// TIA Portal V17 export
// export: Created 2025-03-13T10:30:04.4591601Z, ExportSetting WithDefaults, DisplayName Totally Integrated Automation Portal, DisplayVersion V17 Update 8, DisplayName TIA Portal Openness, DisplayVersion V17 Update 8, DisplayName TIA Portal Version Control Interface, DisplayVersion V17, DisplayName SINAMICS Startdrive Advanced, DisplayVersion V17 SP2, DisplayName SINAMICS Startdrive G110M, G120, G120C, G120D, G120P, G115D, DisplayVersion V17 SP2, DisplayName SINAMICS Startdrive G130, G150, S120, S150, SINAMICS MV, S210, DisplayVersion V17 SP2, DisplayName STEP 7 Professional, DisplayVersion V17 Update 8, DisplayName SINUMERIK ONE STEP 7 Toolbox, DisplayVersion V17 Update 12, DisplayName SINUMERIK 840D sl STEP 7 Toolbox, DisplayVersion V17 Update 12, DisplayName STEP 7 Safety, DisplayVersion V17 Update 6, DisplayName WinCC Advanced, DisplayVersion V17 Update 8
FUNCTION "FC2120_MPP_ITC_IPC" : Void   // FC2120, LAD
{ S7_Optimized_Access := 'FALSE' }
AUTHOR : ETXETAR
VERSION : 1.0
// stored: AutoNumber false, IsIECCheckEnabled false, SetENOAutomatically false, UDAEnableTagReadback false
   VAR_TEMP
      O_BYTE_0 : Struct   // OPTIONS BYTE 0
         IPC : Bool;   // IPC OPTION
      END_STRUCT;
      TCU_INDEX_SEL : Int;
   END_VAR
   VAR CONSTANT
      FC_NUMBER : DInt := 2120;   // FC NUMBER
   END_VAR
   VAR_TEMP   // added for the SCL form of the ladder/FBD networks
      _w1 : Bool;
      _w2 : Bool;
   END_VAR
BEGIN

REGION Network 1: OPTIONS
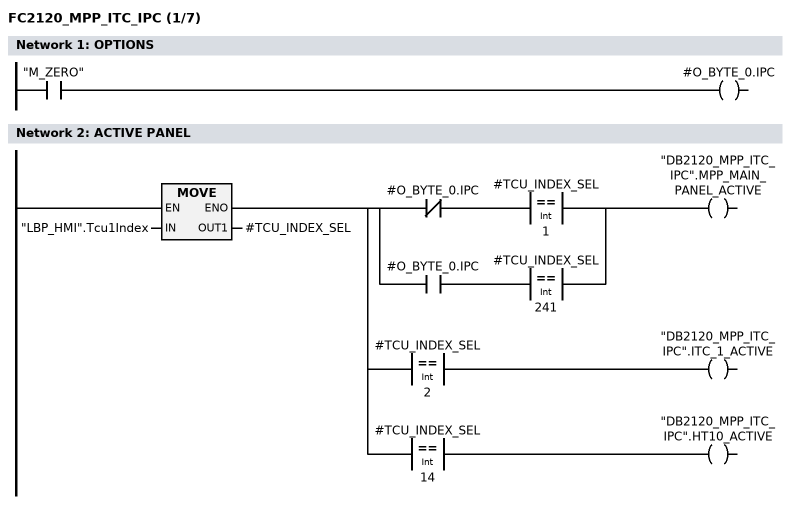
   RUNG wire#powerrail
      Contact( "M_ZERO" )
      Coil( #O_BYTE_0.IPC )
   END_RUNG
   // the same network as SCL:
   #O_BYTE_0.IPC := "M_ZERO";
END_REGION

REGION Network 2: ACTIVE PANEL
   RUNG wire#powerrail
      { S7_GenerateENO := "TRUE" } Move(in := "LBP_HMI".Tcu1Index, out1 => #TCU_INDEX_SEL)
      wire#w1
      I_Contact( #O_BYTE_0.IPC )
      { S7_Templates := "SrcType := Int" } EQ_Contact(in1 := #TCU_INDEX_SEL, in2 := 1)
      wire#w2
      Coil( "DB2120_MPP_ITC_IPC".MPP_MAIN_PANEL_ACTIVE )
   END_RUNG
   RUNG wire#w1
      Contact( #O_BYTE_0.IPC )
      { S7_Templates := "SrcType := Int" } EQ_Contact(in1 := #TCU_INDEX_SEL, in2 := 241)
   END_RUNG wire#w2
   RUNG wire#w1
      { S7_Templates := "SrcType := Int" } EQ_Contact(in1 := #TCU_INDEX_SEL, in2 := 2)
      Coil( "DB2120_MPP_ITC_IPC".ITC_1_ACTIVE )
   END_RUNG
   RUNG wire#w1
      { S7_Templates := "SrcType := Int" } EQ_Contact(in1 := #TCU_INDEX_SEL, in2 := 14)
      Coil( "DB2120_MPP_ITC_IPC".HT10_ACTIVE )
   END_RUNG
   // the same network as SCL:
   // ENO of a box is taken as its EN; it also drops when the box reports an error
   #TCU_INDEX_SEL := "LBP_HMI".Tcu1Index;
   "DB2120_MPP_ITC_IPC".MPP_MAIN_PANEL_ACTIVE := (NOT #O_BYTE_0.IPC AND (#TCU_INDEX_SEL = 1)) OR (#O_BYTE_0.IPC AND (#TCU_INDEX_SEL = 241));
   "DB2120_MPP_ITC_IPC".ITC_1_ACTIVE := #TCU_INDEX_SEL = 2;
   "DB2120_MPP_ITC_IPC".HT10_ACTIVE := #TCU_INDEX_SEL = 14;
END_REGION

REGION Network 3: OVERRIDE
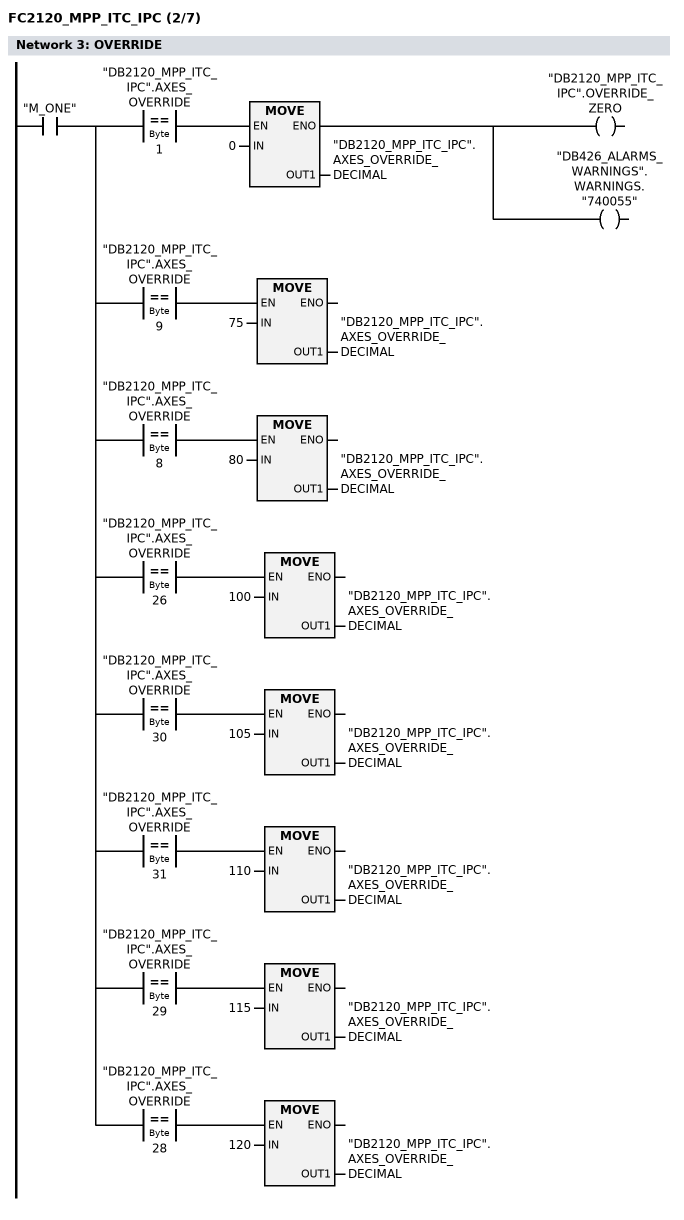
   RUNG wire#powerrail
      Contact( "M_ONE" )
      wire#w1
      { S7_Templates := "SrcType := Byte" } EQ_Contact(in1 := "DB2120_MPP_ITC_IPC".AXES_OVERRIDE, in2 := 1)
      { S7_GenerateENO := "TRUE" } Move(in := 0, out1 => "DB2120_MPP_ITC_IPC".AXES_OVERRIDE_DECIMAL)
      wire#w2
      Coil( "DB2120_MPP_ITC_IPC".OVERRIDE_ZERO )
   END_RUNG
   RUNG wire#w2
      Coil( "DB426_ALARMS_WARNINGS".WARNINGS."740055" )
   END_RUNG
   RUNG wire#w1
      { S7_Templates := "SrcType := Byte" } EQ_Contact(in1 := "DB2120_MPP_ITC_IPC".AXES_OVERRIDE, in2 := 9)
      { S7_GenerateENO := "TRUE" } Move(in := 75, out1 => "DB2120_MPP_ITC_IPC".AXES_OVERRIDE_DECIMAL)
   END_RUNG
   RUNG wire#w1
      { S7_Templates := "SrcType := Byte" } EQ_Contact(in1 := "DB2120_MPP_ITC_IPC".AXES_OVERRIDE, in2 := 8)
      { S7_GenerateENO := "TRUE" } Move(in := 80, out1 => "DB2120_MPP_ITC_IPC".AXES_OVERRIDE_DECIMAL)
   END_RUNG
   RUNG wire#w1
      { S7_Templates := "SrcType := Byte" } EQ_Contact(in1 := "DB2120_MPP_ITC_IPC".AXES_OVERRIDE, in2 := 26)
      { S7_GenerateENO := "TRUE" } Move(in := 100, out1 => "DB2120_MPP_ITC_IPC".AXES_OVERRIDE_DECIMAL)
   END_RUNG
   RUNG wire#w1
      { S7_Templates := "SrcType := Byte" } EQ_Contact(in1 := "DB2120_MPP_ITC_IPC".AXES_OVERRIDE, in2 := 30)
      { S7_GenerateENO := "TRUE" } Move(in := 105, out1 => "DB2120_MPP_ITC_IPC".AXES_OVERRIDE_DECIMAL)
   END_RUNG
   RUNG wire#w1
      { S7_Templates := "SrcType := Byte" } EQ_Contact(in1 := "DB2120_MPP_ITC_IPC".AXES_OVERRIDE, in2 := 31)
      { S7_GenerateENO := "TRUE" } Move(in := 110, out1 => "DB2120_MPP_ITC_IPC".AXES_OVERRIDE_DECIMAL)
   END_RUNG
   RUNG wire#w1
      { S7_Templates := "SrcType := Byte" } EQ_Contact(in1 := "DB2120_MPP_ITC_IPC".AXES_OVERRIDE, in2 := 29)
      { S7_GenerateENO := "TRUE" } Move(in := 115, out1 => "DB2120_MPP_ITC_IPC".AXES_OVERRIDE_DECIMAL)
   END_RUNG
   RUNG wire#w1
      { S7_Templates := "SrcType := Byte" } EQ_Contact(in1 := "DB2120_MPP_ITC_IPC".AXES_OVERRIDE, in2 := 28)
      { S7_GenerateENO := "TRUE" } Move(in := 120, out1 => "DB2120_MPP_ITC_IPC".AXES_OVERRIDE_DECIMAL)
   END_RUNG
   // the same network as SCL:
   // ENO of a box is taken as its EN; it also drops when the box reports an error
   #_w1 := "M_ONE" AND ("DB2120_MPP_ITC_IPC".AXES_OVERRIDE = 1);
   IF #_w1 THEN "DB2120_MPP_ITC_IPC".AXES_OVERRIDE_DECIMAL := 0; END_IF;
   "DB2120_MPP_ITC_IPC".OVERRIDE_ZERO := #_w1;
   "DB426_ALARMS_WARNINGS".WARNINGS."740055" := #_w1;
   IF "M_ONE" AND ("DB2120_MPP_ITC_IPC".AXES_OVERRIDE = 9) THEN
       "DB2120_MPP_ITC_IPC".AXES_OVERRIDE_DECIMAL := 75;
   END_IF;
   IF "M_ONE" AND ("DB2120_MPP_ITC_IPC".AXES_OVERRIDE = 8) THEN
       "DB2120_MPP_ITC_IPC".AXES_OVERRIDE_DECIMAL := 80;
   END_IF;
   IF "M_ONE" AND ("DB2120_MPP_ITC_IPC".AXES_OVERRIDE = 26) THEN
       "DB2120_MPP_ITC_IPC".AXES_OVERRIDE_DECIMAL := 100;
   END_IF;
   IF "M_ONE" AND ("DB2120_MPP_ITC_IPC".AXES_OVERRIDE = 30) THEN
       "DB2120_MPP_ITC_IPC".AXES_OVERRIDE_DECIMAL := 105;
   END_IF;
   IF "M_ONE" AND ("DB2120_MPP_ITC_IPC".AXES_OVERRIDE = 31) THEN
       "DB2120_MPP_ITC_IPC".AXES_OVERRIDE_DECIMAL := 110;
   END_IF;
   IF "M_ONE" AND ("DB2120_MPP_ITC_IPC".AXES_OVERRIDE = 29) THEN
       "DB2120_MPP_ITC_IPC".AXES_OVERRIDE_DECIMAL := 115;
   END_IF;
   IF "M_ONE" AND ("DB2120_MPP_ITC_IPC".AXES_OVERRIDE = 28) THEN
       "DB2120_MPP_ITC_IPC".AXES_OVERRIDE_DECIMAL := 120;
   END_IF;
END_REGION

REGION Network 4: OVERRIDE LOWER THAN 80
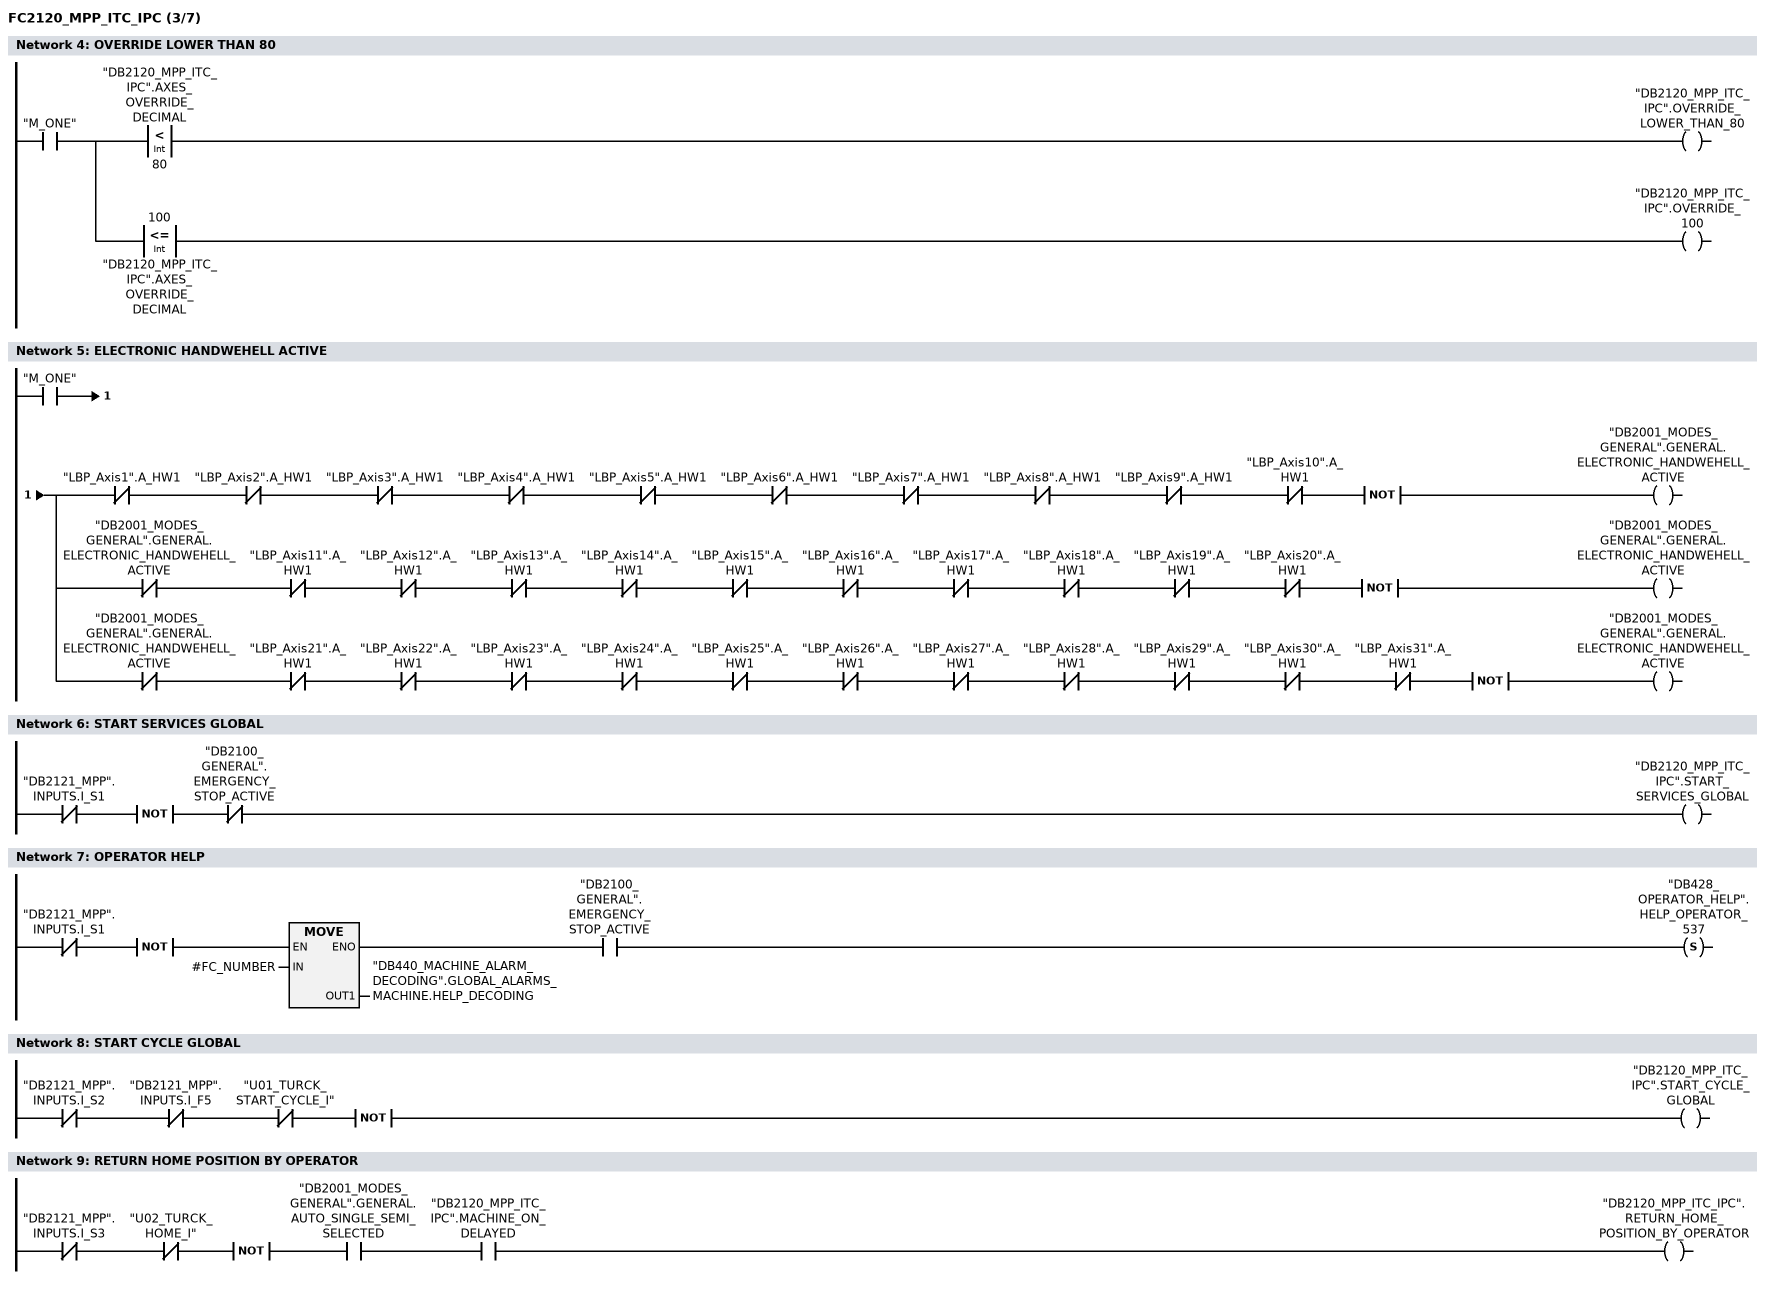
   RUNG wire#powerrail
      Contact( "M_ONE" )
      wire#w1
      { S7_Templates := "SrcType := Int" } LT_Contact(in1 := "DB2120_MPP_ITC_IPC".AXES_OVERRIDE_DECIMAL, in2 := 80)
      Coil( "DB2120_MPP_ITC_IPC".OVERRIDE_LOWER_THAN_80 )
   END_RUNG
   RUNG wire#w1
      { S7_Templates := "SrcType := Int" } LE_Contact(in1 := 100, in2 := "DB2120_MPP_ITC_IPC".AXES_OVERRIDE_DECIMAL)
      Coil( "DB2120_MPP_ITC_IPC".OVERRIDE_100 )
   END_RUNG
   // the same network as SCL:
   "DB2120_MPP_ITC_IPC".OVERRIDE_LOWER_THAN_80 := "M_ONE" AND ("DB2120_MPP_ITC_IPC".AXES_OVERRIDE_DECIMAL < 80);
   "DB2120_MPP_ITC_IPC".OVERRIDE_100 := "M_ONE" AND (100 <= "DB2120_MPP_ITC_IPC".AXES_OVERRIDE_DECIMAL);
END_REGION

REGION Network 5: ELECTRONIC HANDWEHELL ACTIVE
   RUNG wire#powerrail
      Contact( "M_ONE" )
      wire#w1
      I_Contact( "LBP_Axis1".A_HW1 )
      I_Contact( "LBP_Axis2".A_HW1 )
      I_Contact( "LBP_Axis3".A_HW1 )
      I_Contact( "LBP_Axis4".A_HW1 )
      I_Contact( "LBP_Axis5".A_HW1 )
      I_Contact( "LBP_Axis6".A_HW1 )
      I_Contact( "LBP_Axis7".A_HW1 )
      I_Contact( "LBP_Axis8".A_HW1 )
      I_Contact( "LBP_Axis9".A_HW1 )
      I_Contact( "LBP_Axis10".A_HW1 )
      Not()
      Coil( "DB2001_MODES_GENERAL".GENERAL.ELECTRONIC_HANDWEHELL_ACTIVE )
   END_RUNG
   RUNG wire#w1
      I_Contact( "DB2001_MODES_GENERAL".GENERAL.ELECTRONIC_HANDWEHELL_ACTIVE )
      I_Contact( "LBP_Axis11".A_HW1 )
      I_Contact( "LBP_Axis12".A_HW1 )
      I_Contact( "LBP_Axis13".A_HW1 )
      I_Contact( "LBP_Axis14".A_HW1 )
      I_Contact( "LBP_Axis15".A_HW1 )
      I_Contact( "LBP_Axis16".A_HW1 )
      I_Contact( "LBP_Axis17".A_HW1 )
      I_Contact( "LBP_Axis18".A_HW1 )
      I_Contact( "LBP_Axis19".A_HW1 )
      I_Contact( "LBP_Axis20".A_HW1 )
      Not()
      Coil( "DB2001_MODES_GENERAL".GENERAL.ELECTRONIC_HANDWEHELL_ACTIVE )
   END_RUNG
   RUNG wire#w1
      I_Contact( "DB2001_MODES_GENERAL".GENERAL.ELECTRONIC_HANDWEHELL_ACTIVE )
      I_Contact( "LBP_Axis21".A_HW1 )
      I_Contact( "LBP_Axis22".A_HW1 )
      I_Contact( "LBP_Axis23".A_HW1 )
      I_Contact( "LBP_Axis24".A_HW1 )
      I_Contact( "LBP_Axis25".A_HW1 )
      I_Contact( "LBP_Axis26".A_HW1 )
      I_Contact( "LBP_Axis27".A_HW1 )
      I_Contact( "LBP_Axis28".A_HW1 )
      I_Contact( "LBP_Axis29".A_HW1 )
      I_Contact( "LBP_Axis30".A_HW1 )
      I_Contact( "LBP_Axis31".A_HW1 )
      Not()
      Coil( "DB2001_MODES_GENERAL".GENERAL.ELECTRONIC_HANDWEHELL_ACTIVE )
   END_RUNG
   // the same network as SCL:
   "DB2001_MODES_GENERAL".GENERAL.ELECTRONIC_HANDWEHELL_ACTIVE := NOT ("M_ONE" AND NOT "LBP_Axis1".A_HW1 AND NOT "LBP_Axis2".A_HW1 AND NOT "LBP_Axis3".A_HW1 AND NOT "LBP_Axis4".A_HW1 AND NOT "LBP_Axis5".A_HW1 AND NOT "LBP_Axis6".A_HW1 AND NOT "LBP_Axis7".A_HW1 AND NOT "LBP_Axis8".A_HW1 AND NOT "LBP_Axis9".A_HW1 AND NOT "LBP_Axis10".A_HW1);
   "DB2001_MODES_GENERAL".GENERAL.ELECTRONIC_HANDWEHELL_ACTIVE := NOT ("M_ONE" AND NOT "DB2001_MODES_GENERAL".GENERAL.ELECTRONIC_HANDWEHELL_ACTIVE AND NOT "LBP_Axis11".A_HW1 AND NOT "LBP_Axis12".A_HW1 AND NOT "LBP_Axis13".A_HW1 AND NOT "LBP_Axis14".A_HW1 AND NOT "LBP_Axis15".A_HW1 AND NOT "LBP_Axis16".A_HW1 AND NOT "LBP_Axis17".A_HW1 AND NOT "LBP_Axis18".A_HW1 AND NOT "LBP_Axis19".A_HW1 AND NOT "LBP_Axis20".A_HW1);
   "DB2001_MODES_GENERAL".GENERAL.ELECTRONIC_HANDWEHELL_ACTIVE := NOT ("M_ONE" AND NOT "DB2001_MODES_GENERAL".GENERAL.ELECTRONIC_HANDWEHELL_ACTIVE AND NOT "LBP_Axis21".A_HW1 AND NOT "LBP_Axis22".A_HW1 AND NOT "LBP_Axis23".A_HW1 AND NOT "LBP_Axis24".A_HW1 AND NOT "LBP_Axis25".A_HW1 AND NOT "LBP_Axis26".A_HW1 AND NOT "LBP_Axis27".A_HW1 AND NOT "LBP_Axis28".A_HW1 AND NOT "LBP_Axis29".A_HW1 AND NOT "LBP_Axis30".A_HW1 AND NOT "LBP_Axis31".A_HW1);
END_REGION

REGION Network 6: START SERVICES GLOBAL
   RUNG wire#powerrail
      I_Contact( "DB2121_MPP".INPUTS.I_S1 )
      Not()
      I_Contact( "DB2100_GENERAL".EMERGENCY_STOP_ACTIVE )
      Coil( "DB2120_MPP_ITC_IPC".START_SERVICES_GLOBAL )
   END_RUNG
   // the same network as SCL:
   "DB2120_MPP_ITC_IPC".START_SERVICES_GLOBAL := NOT (NOT "DB2121_MPP".INPUTS.I_S1) AND NOT "DB2100_GENERAL".EMERGENCY_STOP_ACTIVE;
END_REGION

REGION Network 7: OPERATOR HELP
   RUNG wire#powerrail
      I_Contact( "DB2121_MPP".INPUTS.I_S1 )
      Not()
      { S7_GenerateENO := "TRUE" } Move(in := #FC_NUMBER, out1 => "DB440_MACHINE_ALARM_DECODING".GLOBAL_ALARMS_MACHINE.HELP_DECODING)
      Contact( "DB2100_GENERAL".EMERGENCY_STOP_ACTIVE )
      S_Coil( "DB428_OPERATOR_HELP".HELP_OPERATOR_537 )
   END_RUNG
   // the same network as SCL:
   // ENO of a box is taken as its EN; it also drops when the box reports an error
   #_w1 := NOT (NOT "DB2121_MPP".INPUTS.I_S1);
   IF #_w1 THEN "DB440_MACHINE_ALARM_DECODING".GLOBAL_ALARMS_MACHINE.HELP_DECODING := #FC_NUMBER; END_IF;
   IF #_w1 AND "DB2100_GENERAL".EMERGENCY_STOP_ACTIVE THEN
       "DB428_OPERATOR_HELP".HELP_OPERATOR_537 := TRUE;
   END_IF;
END_REGION

REGION Network 8: START CYCLE GLOBAL
   RUNG wire#powerrail
      I_Contact( "DB2121_MPP".INPUTS.I_S2 )
      I_Contact( "DB2121_MPP".INPUTS.I_F5 )
      I_Contact( "U01_TURCK_START_CYCLE_I" )
      Not()
      Coil( "DB2120_MPP_ITC_IPC".START_CYCLE_GLOBAL )
   END_RUNG
   // the same network as SCL:
   "DB2120_MPP_ITC_IPC".START_CYCLE_GLOBAL := NOT (NOT "DB2121_MPP".INPUTS.I_S2 AND NOT "DB2121_MPP".INPUTS.I_F5 AND NOT "U01_TURCK_START_CYCLE_I");
END_REGION

REGION Network 9: RETURN HOME POSITION BY OPERATOR
   RUNG wire#powerrail
      I_Contact( "DB2121_MPP".INPUTS.I_S3 )
      I_Contact( "U02_TURCK_HOME_I" )
      Not()
      Contact( "DB2001_MODES_GENERAL".GENERAL.AUTO_SINGLE_SEMI_SELECTED )
      Contact( "DB2120_MPP_ITC_IPC".MACHINE_ON_DELAYED )
      Coil( "DB2120_MPP_ITC_IPC".RETURN_HOME_POSITION_BY_OPERATOR )
   END_RUNG
   // the same network as SCL:
   "DB2120_MPP_ITC_IPC".RETURN_HOME_POSITION_BY_OPERATOR := NOT (NOT "DB2121_MPP".INPUTS.I_S3 AND NOT "U02_TURCK_HOME_I") AND "DB2001_MODES_GENERAL".GENERAL.AUTO_SINGLE_SEMI_SELECTED AND "DB2120_MPP_ITC_IPC".MACHINE_ON_DELAYED;
END_REGION

REGION Network 10: RETURN HOME POSITION FROM MPP-AUX PANEL
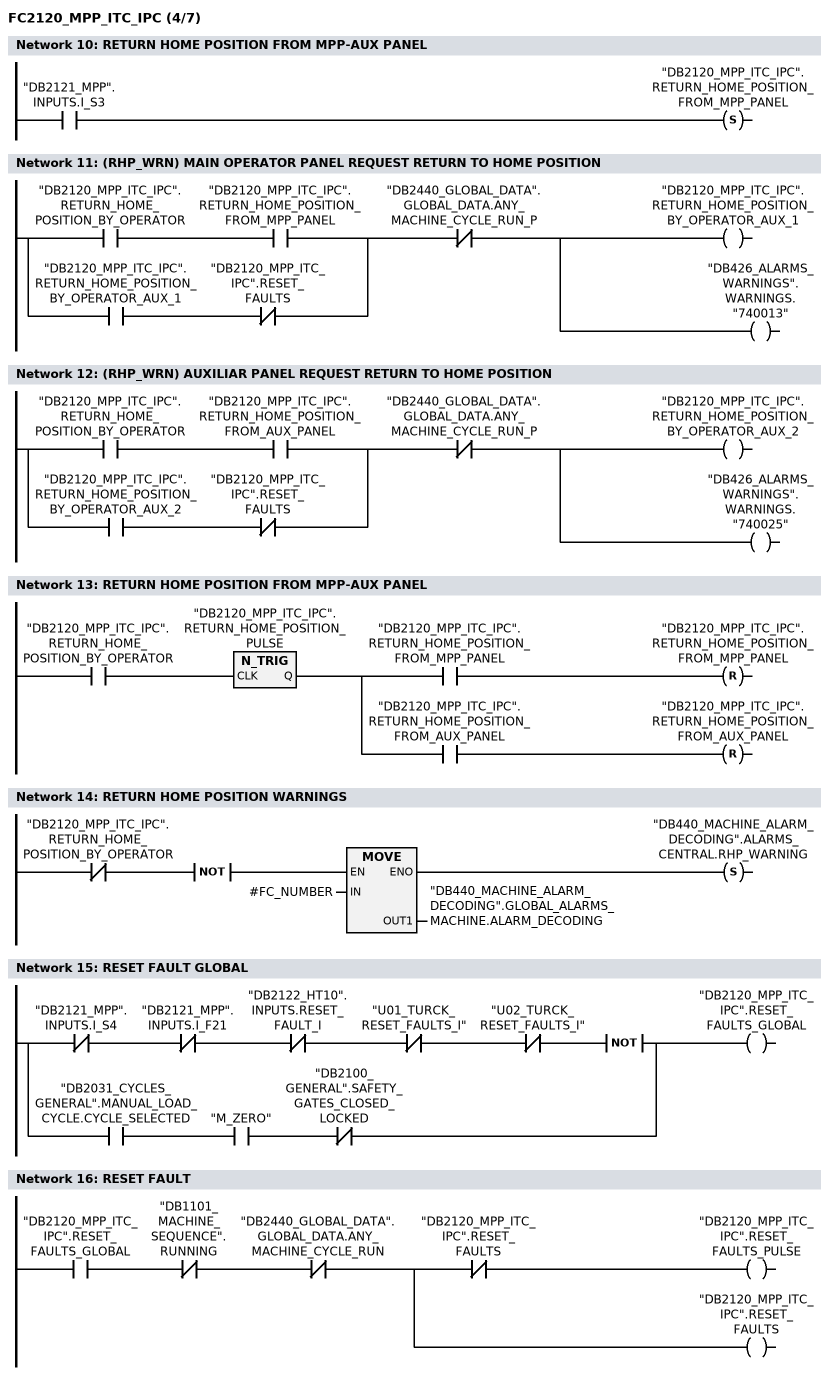
   RUNG wire#powerrail
      Contact( "DB2121_MPP".INPUTS.I_S3 )
      S_Coil( "DB2120_MPP_ITC_IPC".RETURN_HOME_POSITION_FROM_MPP_PANEL )
   END_RUNG
   // the same network as SCL:
   IF "DB2121_MPP".INPUTS.I_S3 THEN "DB2120_MPP_ITC_IPC".RETURN_HOME_POSITION_FROM_MPP_PANEL := TRUE; END_IF;
END_REGION

REGION Network 11: (RHP_WRN) MAIN OPERATOR PANEL REQUEST RETURN TO HOME POSITION
   RUNG wire#powerrail
      Contact( "DB2120_MPP_ITC_IPC".RETURN_HOME_POSITION_BY_OPERATOR )
      Contact( "DB2120_MPP_ITC_IPC".RETURN_HOME_POSITION_FROM_MPP_PANEL )
      wire#w1
      I_Contact( "DB2440_GLOBAL_DATA".GLOBAL_DATA.ANY_MACHINE_CYCLE_RUN_P )
      wire#w2
      Coil( "DB2120_MPP_ITC_IPC".RETURN_HOME_POSITION_BY_OPERATOR_AUX_1 )
   END_RUNG
   RUNG wire#powerrail
      Contact( "DB2120_MPP_ITC_IPC".RETURN_HOME_POSITION_BY_OPERATOR_AUX_1 )
      I_Contact( "DB2120_MPP_ITC_IPC".RESET_FAULTS )
   END_RUNG wire#w1
   RUNG wire#w2
      Coil( "DB426_ALARMS_WARNINGS".WARNINGS."740013" )
   END_RUNG
   // the same network as SCL:
   "DB2120_MPP_ITC_IPC".RETURN_HOME_POSITION_BY_OPERATOR_AUX_1 := (("DB2120_MPP_ITC_IPC".RETURN_HOME_POSITION_BY_OPERATOR AND "DB2120_MPP_ITC_IPC".RETURN_HOME_POSITION_FROM_MPP_PANEL) OR ("DB2120_MPP_ITC_IPC".RETURN_HOME_POSITION_BY_OPERATOR_AUX_1 AND NOT "DB2120_MPP_ITC_IPC".RESET_FAULTS)) AND NOT "DB2440_GLOBAL_DATA".GLOBAL_DATA.ANY_MACHINE_CYCLE_RUN_P;
   "DB426_ALARMS_WARNINGS".WARNINGS."740013" := "DB2120_MPP_ITC_IPC".RETURN_HOME_POSITION_BY_OPERATOR_AUX_1;
END_REGION

REGION Network 12: (RHP_WRN) AUXILIAR PANEL REQUEST RETURN TO HOME POSITION
   RUNG wire#powerrail
      Contact( "DB2120_MPP_ITC_IPC".RETURN_HOME_POSITION_BY_OPERATOR )
      Contact( "DB2120_MPP_ITC_IPC".RETURN_HOME_POSITION_FROM_AUX_PANEL )
      wire#w1
      I_Contact( "DB2440_GLOBAL_DATA".GLOBAL_DATA.ANY_MACHINE_CYCLE_RUN_P )
      wire#w2
      Coil( "DB2120_MPP_ITC_IPC".RETURN_HOME_POSITION_BY_OPERATOR_AUX_2 )
   END_RUNG
   RUNG wire#powerrail
      Contact( "DB2120_MPP_ITC_IPC".RETURN_HOME_POSITION_BY_OPERATOR_AUX_2 )
      I_Contact( "DB2120_MPP_ITC_IPC".RESET_FAULTS )
   END_RUNG wire#w1
   RUNG wire#w2
      Coil( "DB426_ALARMS_WARNINGS".WARNINGS."740025" )
   END_RUNG
   // the same network as SCL:
   "DB2120_MPP_ITC_IPC".RETURN_HOME_POSITION_BY_OPERATOR_AUX_2 := (("DB2120_MPP_ITC_IPC".RETURN_HOME_POSITION_BY_OPERATOR AND "DB2120_MPP_ITC_IPC".RETURN_HOME_POSITION_FROM_AUX_PANEL) OR ("DB2120_MPP_ITC_IPC".RETURN_HOME_POSITION_BY_OPERATOR_AUX_2 AND NOT "DB2120_MPP_ITC_IPC".RESET_FAULTS)) AND NOT "DB2440_GLOBAL_DATA".GLOBAL_DATA.ANY_MACHINE_CYCLE_RUN_P;
   "DB426_ALARMS_WARNINGS".WARNINGS."740025" := "DB2120_MPP_ITC_IPC".RETURN_HOME_POSITION_BY_OPERATOR_AUX_2;
END_REGION

REGION Network 13: RETURN HOME POSITION FROM MPP-AUX PANEL
   RUNG wire#powerrail
      Contact( "DB2120_MPP_ITC_IPC".RETURN_HOME_POSITION_BY_OPERATOR )
      N_Trig( "DB2120_MPP_ITC_IPC".RETURN_HOME_POSITION_PULSE )
      wire#w1
      Contact( "DB2120_MPP_ITC_IPC".RETURN_HOME_POSITION_FROM_MPP_PANEL )
      R_Coil( "DB2120_MPP_ITC_IPC".RETURN_HOME_POSITION_FROM_MPP_PANEL )
   END_RUNG
   RUNG wire#w1
      Contact( "DB2120_MPP_ITC_IPC".RETURN_HOME_POSITION_FROM_AUX_PANEL )
      R_Coil( "DB2120_MPP_ITC_IPC".RETURN_HOME_POSITION_FROM_AUX_PANEL )
   END_RUNG
   // the same network as SCL:
   #_w1 := NOT "DB2120_MPP_ITC_IPC".RETURN_HOME_POSITION_BY_OPERATOR AND "DB2120_MPP_ITC_IPC".RETURN_HOME_POSITION_PULSE;   // falling edge
   "DB2120_MPP_ITC_IPC".RETURN_HOME_POSITION_PULSE := "DB2120_MPP_ITC_IPC".RETURN_HOME_POSITION_BY_OPERATOR;
   IF #_w1 AND "DB2120_MPP_ITC_IPC".RETURN_HOME_POSITION_FROM_MPP_PANEL THEN
       "DB2120_MPP_ITC_IPC".RETURN_HOME_POSITION_FROM_MPP_PANEL := FALSE;
   END_IF;
   IF #_w1 AND "DB2120_MPP_ITC_IPC".RETURN_HOME_POSITION_FROM_AUX_PANEL THEN
       "DB2120_MPP_ITC_IPC".RETURN_HOME_POSITION_FROM_AUX_PANEL := FALSE;
   END_IF;
END_REGION

REGION Network 14: RETURN HOME POSITION WARNINGS
   RUNG wire#powerrail
      I_Contact( "DB2120_MPP_ITC_IPC".RETURN_HOME_POSITION_BY_OPERATOR )
      Not()
      { S7_GenerateENO := "TRUE" } Move(in := #FC_NUMBER, out1 => "DB440_MACHINE_ALARM_DECODING".GLOBAL_ALARMS_MACHINE.ALARM_DECODING)
      S_Coil( "DB440_MACHINE_ALARM_DECODING".ALARMS_CENTRAL.RHP_WARNING )
   END_RUNG
   // the same network as SCL:
   // ENO of a box is taken as its EN; it also drops when the box reports an error
   IF NOT (NOT "DB2120_MPP_ITC_IPC".RETURN_HOME_POSITION_BY_OPERATOR) THEN
       "DB440_MACHINE_ALARM_DECODING".GLOBAL_ALARMS_MACHINE.ALARM_DECODING := #FC_NUMBER;
       "DB440_MACHINE_ALARM_DECODING".ALARMS_CENTRAL.RHP_WARNING := TRUE;
   END_IF;
END_REGION

REGION Network 15: RESET FAULT GLOBAL
   RUNG wire#powerrail
      I_Contact( "DB2121_MPP".INPUTS.I_S4 )
      I_Contact( "DB2121_MPP".INPUTS.I_F21 )
      I_Contact( "DB2122_HT10".INPUTS.RESET_FAULT_I )
      I_Contact( "U01_TURCK_RESET_FAULTS_I" )
      I_Contact( "U02_TURCK_RESET_FAULTS_I" )
      Not()
      wire#w1
      Coil( "DB2120_MPP_ITC_IPC".RESET_FAULTS_GLOBAL )
   END_RUNG
   RUNG wire#powerrail
      Contact( "DB2031_CYCLES_GENERAL".MANUAL_LOAD_CYCLE.CYCLE_SELECTED )
      Contact( "M_ZERO" )
      I_Contact( "DB2100_GENERAL".SAFETY_GATES_CLOSED_LOCKED )
   END_RUNG wire#w1
   // the same network as SCL:
   "DB2120_MPP_ITC_IPC".RESET_FAULTS_GLOBAL := NOT (NOT "DB2121_MPP".INPUTS.I_S4 AND NOT "DB2121_MPP".INPUTS.I_F21 AND NOT "DB2122_HT10".INPUTS.RESET_FAULT_I AND NOT "U01_TURCK_RESET_FAULTS_I" AND NOT "U02_TURCK_RESET_FAULTS_I") OR ("DB2031_CYCLES_GENERAL".MANUAL_LOAD_CYCLE.CYCLE_SELECTED AND "M_ZERO" AND NOT "DB2100_GENERAL".SAFETY_GATES_CLOSED_LOCKED);
END_REGION

REGION Network 16: RESET FAULT
   RUNG wire#powerrail
      Contact( "DB2120_MPP_ITC_IPC".RESET_FAULTS_GLOBAL )
      I_Contact( "DB1101_MACHINE_SEQUENCE".RUNNING )
      I_Contact( "DB2440_GLOBAL_DATA".GLOBAL_DATA.ANY_MACHINE_CYCLE_RUN )
      wire#w1
      I_Contact( "DB2120_MPP_ITC_IPC".RESET_FAULTS )
      Coil( "DB2120_MPP_ITC_IPC".RESET_FAULTS_PULSE )
   END_RUNG
   RUNG wire#w1
      Coil( "DB2120_MPP_ITC_IPC".RESET_FAULTS )
   END_RUNG
   // the same network as SCL:
   #_w1 := "DB2120_MPP_ITC_IPC".RESET_FAULTS_GLOBAL AND NOT "DB1101_MACHINE_SEQUENCE".RUNNING AND NOT "DB2440_GLOBAL_DATA".GLOBAL_DATA.ANY_MACHINE_CYCLE_RUN;
   "DB2120_MPP_ITC_IPC".RESET_FAULTS_PULSE := #_w1 AND NOT "DB2120_MPP_ITC_IPC".RESET_FAULTS;
   "DB2120_MPP_ITC_IPC".RESET_FAULTS := #_w1;
END_REGION

REGION Network 17: STOP SERVICES GLOBAL
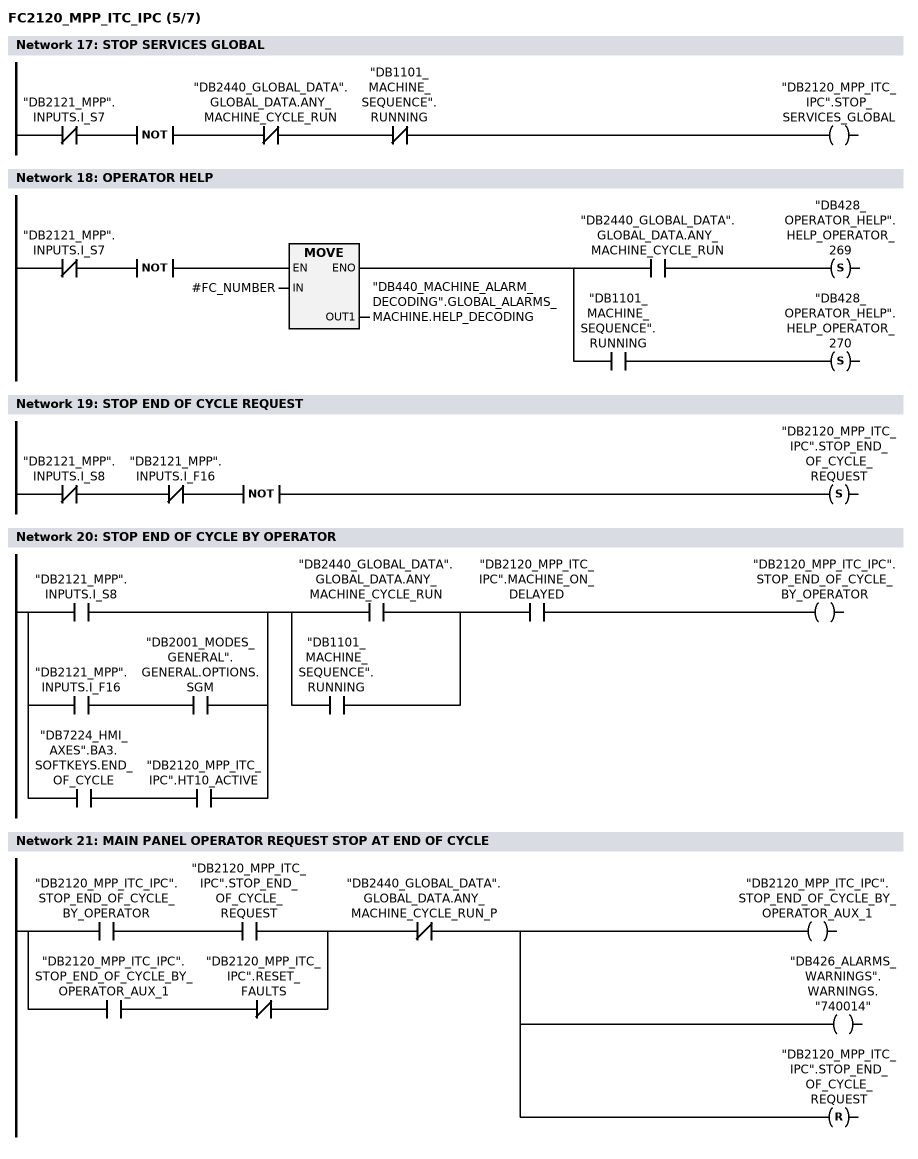
   RUNG wire#powerrail
      I_Contact( "DB2121_MPP".INPUTS.I_S7 )
      Not()
      I_Contact( "DB2440_GLOBAL_DATA".GLOBAL_DATA.ANY_MACHINE_CYCLE_RUN )
      I_Contact( "DB1101_MACHINE_SEQUENCE".RUNNING )
      Coil( "DB2120_MPP_ITC_IPC".STOP_SERVICES_GLOBAL )
   END_RUNG
   // the same network as SCL:
   "DB2120_MPP_ITC_IPC".STOP_SERVICES_GLOBAL := NOT (NOT "DB2121_MPP".INPUTS.I_S7) AND NOT "DB2440_GLOBAL_DATA".GLOBAL_DATA.ANY_MACHINE_CYCLE_RUN AND NOT "DB1101_MACHINE_SEQUENCE".RUNNING;
END_REGION

REGION Network 18: OPERATOR HELP
   RUNG wire#powerrail
      I_Contact( "DB2121_MPP".INPUTS.I_S7 )
      Not()
      { S7_GenerateENO := "TRUE" } Move(in := #FC_NUMBER, out1 => "DB440_MACHINE_ALARM_DECODING".GLOBAL_ALARMS_MACHINE.HELP_DECODING)
      wire#w1
      Contact( "DB2440_GLOBAL_DATA".GLOBAL_DATA.ANY_MACHINE_CYCLE_RUN )
      S_Coil( "DB428_OPERATOR_HELP".HELP_OPERATOR_269 )
   END_RUNG
   RUNG wire#w1
      Contact( "DB1101_MACHINE_SEQUENCE".RUNNING )
      S_Coil( "DB428_OPERATOR_HELP".HELP_OPERATOR_270 )
   END_RUNG
   // the same network as SCL:
   // ENO of a box is taken as its EN; it also drops when the box reports an error
   #_w1 := NOT (NOT "DB2121_MPP".INPUTS.I_S7);
   IF #_w1 THEN "DB440_MACHINE_ALARM_DECODING".GLOBAL_ALARMS_MACHINE.HELP_DECODING := #FC_NUMBER; END_IF;
   IF #_w1 AND "DB2440_GLOBAL_DATA".GLOBAL_DATA.ANY_MACHINE_CYCLE_RUN THEN
       "DB428_OPERATOR_HELP".HELP_OPERATOR_269 := TRUE;
   END_IF;
   IF #_w1 AND "DB1101_MACHINE_SEQUENCE".RUNNING THEN
       "DB428_OPERATOR_HELP".HELP_OPERATOR_270 := TRUE;
   END_IF;
END_REGION

REGION Network 19: STOP END OF CYCLE REQUEST
   RUNG wire#powerrail
      I_Contact( "DB2121_MPP".INPUTS.I_S8 )
      I_Contact( "DB2121_MPP".INPUTS.I_F16 )
      Not()
      S_Coil( "DB2120_MPP_ITC_IPC".STOP_END_OF_CYCLE_REQUEST )
   END_RUNG
   // the same network as SCL:
   IF NOT (NOT "DB2121_MPP".INPUTS.I_S8 AND NOT "DB2121_MPP".INPUTS.I_F16) THEN
       "DB2120_MPP_ITC_IPC".STOP_END_OF_CYCLE_REQUEST := TRUE;
   END_IF;
END_REGION

REGION Network 20: STOP END OF CYCLE BY OPERATOR
   RUNG wire#powerrail
      Contact( "DB2121_MPP".INPUTS.I_S8 )
      wire#w1
      Contact( "DB2440_GLOBAL_DATA".GLOBAL_DATA.ANY_MACHINE_CYCLE_RUN )
      wire#w2
      Contact( "DB2120_MPP_ITC_IPC".MACHINE_ON_DELAYED )
      Coil( "DB2120_MPP_ITC_IPC".STOP_END_OF_CYCLE_BY_OPERATOR )
   END_RUNG
   RUNG wire#powerrail
      Contact( "DB2121_MPP".INPUTS.I_F16 )
      Contact( "DB2001_MODES_GENERAL".GENERAL.OPTIONS.SGM )
   END_RUNG wire#w1
   RUNG wire#powerrail
      Contact( "DB7224_HMI_AXES".BA3.SOFTKEYS.END_OF_CYCLE )
      Contact( "DB2120_MPP_ITC_IPC".HT10_ACTIVE )
   END_RUNG wire#w1
   RUNG wire#w1
      Contact( "DB1101_MACHINE_SEQUENCE".RUNNING )
   END_RUNG wire#w2
   // the same network as SCL:
   "DB2120_MPP_ITC_IPC".STOP_END_OF_CYCLE_BY_OPERATOR := ("DB2121_MPP".INPUTS.I_S8 OR ("DB2121_MPP".INPUTS.I_F16 AND "DB2001_MODES_GENERAL".GENERAL.OPTIONS.SGM) OR ("DB7224_HMI_AXES".BA3.SOFTKEYS.END_OF_CYCLE AND "DB2120_MPP_ITC_IPC".HT10_ACTIVE)) AND ("DB2440_GLOBAL_DATA".GLOBAL_DATA.ANY_MACHINE_CYCLE_RUN OR "DB1101_MACHINE_SEQUENCE".RUNNING) AND "DB2120_MPP_ITC_IPC".MACHINE_ON_DELAYED;
END_REGION

REGION Network 21: MAIN PANEL OPERATOR REQUEST STOP AT END OF CYCLE
   RUNG wire#powerrail
      Contact( "DB2120_MPP_ITC_IPC".STOP_END_OF_CYCLE_BY_OPERATOR )
      Contact( "DB2120_MPP_ITC_IPC".STOP_END_OF_CYCLE_REQUEST )
      wire#w1
      I_Contact( "DB2440_GLOBAL_DATA".GLOBAL_DATA.ANY_MACHINE_CYCLE_RUN_P )
      wire#w2
      Coil( "DB2120_MPP_ITC_IPC".STOP_END_OF_CYCLE_BY_OPERATOR_AUX_1 )
   END_RUNG
   RUNG wire#powerrail
      Contact( "DB2120_MPP_ITC_IPC".STOP_END_OF_CYCLE_BY_OPERATOR_AUX_1 )
      I_Contact( "DB2120_MPP_ITC_IPC".RESET_FAULTS )
   END_RUNG wire#w1
   RUNG wire#w2
      Coil( "DB426_ALARMS_WARNINGS".WARNINGS."740014" )
   END_RUNG
   RUNG wire#w2
      R_Coil( "DB2120_MPP_ITC_IPC".STOP_END_OF_CYCLE_REQUEST )
   END_RUNG
   // the same network as SCL:
   "DB2120_MPP_ITC_IPC".STOP_END_OF_CYCLE_BY_OPERATOR_AUX_1 := (("DB2120_MPP_ITC_IPC".STOP_END_OF_CYCLE_BY_OPERATOR AND "DB2120_MPP_ITC_IPC".STOP_END_OF_CYCLE_REQUEST) OR ("DB2120_MPP_ITC_IPC".STOP_END_OF_CYCLE_BY_OPERATOR_AUX_1 AND NOT "DB2120_MPP_ITC_IPC".RESET_FAULTS)) AND NOT "DB2440_GLOBAL_DATA".GLOBAL_DATA.ANY_MACHINE_CYCLE_RUN_P;
   "DB426_ALARMS_WARNINGS".WARNINGS."740014" := "DB2120_MPP_ITC_IPC".STOP_END_OF_CYCLE_BY_OPERATOR_AUX_1;
   IF "DB2120_MPP_ITC_IPC".STOP_END_OF_CYCLE_BY_OPERATOR_AUX_1 THEN
       "DB2120_MPP_ITC_IPC".STOP_END_OF_CYCLE_REQUEST := FALSE;
   END_IF;
END_REGION

REGION Network 22: AUXILIARY PANEL OPERATOR REQUEST STOP AT END OF CYCLE
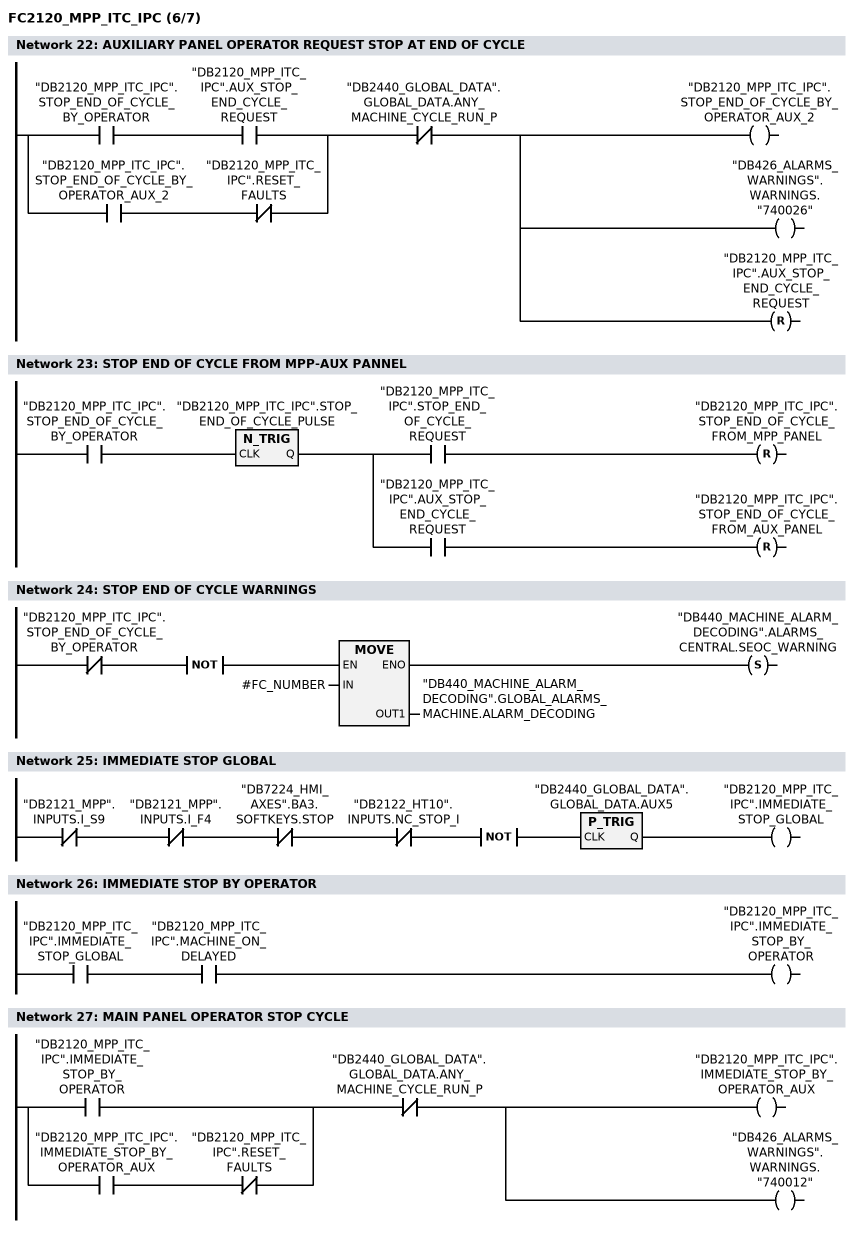
   RUNG wire#powerrail
      Contact( "DB2120_MPP_ITC_IPC".STOP_END_OF_CYCLE_BY_OPERATOR )
      Contact( "DB2120_MPP_ITC_IPC".AUX_STOP_END_CYCLE_REQUEST )
      wire#w1
      I_Contact( "DB2440_GLOBAL_DATA".GLOBAL_DATA.ANY_MACHINE_CYCLE_RUN_P )
      wire#w2
      Coil( "DB2120_MPP_ITC_IPC".STOP_END_OF_CYCLE_BY_OPERATOR_AUX_2 )
   END_RUNG
   RUNG wire#powerrail
      Contact( "DB2120_MPP_ITC_IPC".STOP_END_OF_CYCLE_BY_OPERATOR_AUX_2 )
      I_Contact( "DB2120_MPP_ITC_IPC".RESET_FAULTS )
   END_RUNG wire#w1
   RUNG wire#w2
      Coil( "DB426_ALARMS_WARNINGS".WARNINGS."740026" )
   END_RUNG
   RUNG wire#w2
      R_Coil( "DB2120_MPP_ITC_IPC".AUX_STOP_END_CYCLE_REQUEST )
   END_RUNG
   // the same network as SCL:
   "DB2120_MPP_ITC_IPC".STOP_END_OF_CYCLE_BY_OPERATOR_AUX_2 := (("DB2120_MPP_ITC_IPC".STOP_END_OF_CYCLE_BY_OPERATOR AND "DB2120_MPP_ITC_IPC".AUX_STOP_END_CYCLE_REQUEST) OR ("DB2120_MPP_ITC_IPC".STOP_END_OF_CYCLE_BY_OPERATOR_AUX_2 AND NOT "DB2120_MPP_ITC_IPC".RESET_FAULTS)) AND NOT "DB2440_GLOBAL_DATA".GLOBAL_DATA.ANY_MACHINE_CYCLE_RUN_P;
   "DB426_ALARMS_WARNINGS".WARNINGS."740026" := "DB2120_MPP_ITC_IPC".STOP_END_OF_CYCLE_BY_OPERATOR_AUX_2;
   IF "DB2120_MPP_ITC_IPC".STOP_END_OF_CYCLE_BY_OPERATOR_AUX_2 THEN
       "DB2120_MPP_ITC_IPC".AUX_STOP_END_CYCLE_REQUEST := FALSE;
   END_IF;
END_REGION

REGION Network 23: STOP END OF CYCLE FROM MPP-AUX PANNEL
   RUNG wire#powerrail
      Contact( "DB2120_MPP_ITC_IPC".STOP_END_OF_CYCLE_BY_OPERATOR )
      N_Trig( "DB2120_MPP_ITC_IPC".STOP_END_OF_CYCLE_PULSE )
      wire#w1
      Contact( "DB2120_MPP_ITC_IPC".STOP_END_OF_CYCLE_REQUEST )
      R_Coil( "DB2120_MPP_ITC_IPC".STOP_END_OF_CYCLE_FROM_MPP_PANEL )
   END_RUNG
   RUNG wire#w1
      Contact( "DB2120_MPP_ITC_IPC".AUX_STOP_END_CYCLE_REQUEST )
      R_Coil( "DB2120_MPP_ITC_IPC".STOP_END_OF_CYCLE_FROM_AUX_PANEL )
   END_RUNG
   // the same network as SCL:
   #_w1 := NOT "DB2120_MPP_ITC_IPC".STOP_END_OF_CYCLE_BY_OPERATOR AND "DB2120_MPP_ITC_IPC".STOP_END_OF_CYCLE_PULSE;   // falling edge
   "DB2120_MPP_ITC_IPC".STOP_END_OF_CYCLE_PULSE := "DB2120_MPP_ITC_IPC".STOP_END_OF_CYCLE_BY_OPERATOR;
   IF #_w1 AND "DB2120_MPP_ITC_IPC".STOP_END_OF_CYCLE_REQUEST THEN
       "DB2120_MPP_ITC_IPC".STOP_END_OF_CYCLE_FROM_MPP_PANEL := FALSE;
   END_IF;
   IF #_w1 AND "DB2120_MPP_ITC_IPC".AUX_STOP_END_CYCLE_REQUEST THEN
       "DB2120_MPP_ITC_IPC".STOP_END_OF_CYCLE_FROM_AUX_PANEL := FALSE;
   END_IF;
END_REGION

REGION Network 24: STOP END OF CYCLE WARNINGS
   RUNG wire#powerrail
      I_Contact( "DB2120_MPP_ITC_IPC".STOP_END_OF_CYCLE_BY_OPERATOR )
      Not()
      { S7_GenerateENO := "TRUE" } Move(in := #FC_NUMBER, out1 => "DB440_MACHINE_ALARM_DECODING".GLOBAL_ALARMS_MACHINE.ALARM_DECODING)
      S_Coil( "DB440_MACHINE_ALARM_DECODING".ALARMS_CENTRAL.SEOC_WARNING )
   END_RUNG
   // the same network as SCL:
   // ENO of a box is taken as its EN; it also drops when the box reports an error
   IF NOT (NOT "DB2120_MPP_ITC_IPC".STOP_END_OF_CYCLE_BY_OPERATOR) THEN
       "DB440_MACHINE_ALARM_DECODING".GLOBAL_ALARMS_MACHINE.ALARM_DECODING := #FC_NUMBER;
       "DB440_MACHINE_ALARM_DECODING".ALARMS_CENTRAL.SEOC_WARNING := TRUE;
   END_IF;
END_REGION

REGION Network 25: IMMEDIATE STOP GLOBAL
   RUNG wire#powerrail
      I_Contact( "DB2121_MPP".INPUTS.I_S9 )
      I_Contact( "DB2121_MPP".INPUTS.I_F4 )
      I_Contact( "DB7224_HMI_AXES".BA3.SOFTKEYS.STOP )
      I_Contact( "DB2122_HT10".INPUTS.NC_STOP_I )
      Not()
      P_Trig( "DB2440_GLOBAL_DATA".GLOBAL_DATA.AUX5 )
      Coil( "DB2120_MPP_ITC_IPC".IMMEDIATE_STOP_GLOBAL )
   END_RUNG
   // the same network as SCL:
   #_w1 := NOT (NOT "DB2121_MPP".INPUTS.I_S9 AND NOT "DB2121_MPP".INPUTS.I_F4 AND NOT "DB7224_HMI_AXES".BA3.SOFTKEYS.STOP AND NOT "DB2122_HT10".INPUTS.NC_STOP_I);
   #_w2 := #_w1 AND NOT "DB2440_GLOBAL_DATA".GLOBAL_DATA.AUX5;   // rising edge
   "DB2440_GLOBAL_DATA".GLOBAL_DATA.AUX5 := #_w1;
   "DB2120_MPP_ITC_IPC".IMMEDIATE_STOP_GLOBAL := #_w2;
END_REGION

REGION Network 26: IMMEDIATE STOP BY OPERATOR
   RUNG wire#powerrail
      Contact( "DB2120_MPP_ITC_IPC".IMMEDIATE_STOP_GLOBAL )
      Contact( "DB2120_MPP_ITC_IPC".MACHINE_ON_DELAYED )
      Coil( "DB2120_MPP_ITC_IPC".IMMEDIATE_STOP_BY_OPERATOR )
   END_RUNG
   // the same network as SCL:
   "DB2120_MPP_ITC_IPC".IMMEDIATE_STOP_BY_OPERATOR := "DB2120_MPP_ITC_IPC".IMMEDIATE_STOP_GLOBAL AND "DB2120_MPP_ITC_IPC".MACHINE_ON_DELAYED;
END_REGION

REGION Network 27: MAIN PANEL OPERATOR STOP CYCLE
   RUNG wire#powerrail
      Contact( "DB2120_MPP_ITC_IPC".IMMEDIATE_STOP_BY_OPERATOR )
      wire#w1
      I_Contact( "DB2440_GLOBAL_DATA".GLOBAL_DATA.ANY_MACHINE_CYCLE_RUN_P )
      wire#w2
      Coil( "DB2120_MPP_ITC_IPC".IMMEDIATE_STOP_BY_OPERATOR_AUX )
   END_RUNG
   RUNG wire#powerrail
      Contact( "DB2120_MPP_ITC_IPC".IMMEDIATE_STOP_BY_OPERATOR_AUX )
      I_Contact( "DB2120_MPP_ITC_IPC".RESET_FAULTS )
   END_RUNG wire#w1
   RUNG wire#w2
      Coil( "DB426_ALARMS_WARNINGS".WARNINGS."740012" )
   END_RUNG
   // the same network as SCL:
   "DB2120_MPP_ITC_IPC".IMMEDIATE_STOP_BY_OPERATOR_AUX := ("DB2120_MPP_ITC_IPC".IMMEDIATE_STOP_BY_OPERATOR OR ("DB2120_MPP_ITC_IPC".IMMEDIATE_STOP_BY_OPERATOR_AUX AND NOT "DB2120_MPP_ITC_IPC".RESET_FAULTS)) AND NOT "DB2440_GLOBAL_DATA".GLOBAL_DATA.ANY_MACHINE_CYCLE_RUN_P;
   "DB426_ALARMS_WARNINGS".WARNINGS."740012" := "DB2120_MPP_ITC_IPC".IMMEDIATE_STOP_BY_OPERATOR_AUX;
END_REGION

REGION Network 28: IMMEDIATE STOP WARNING
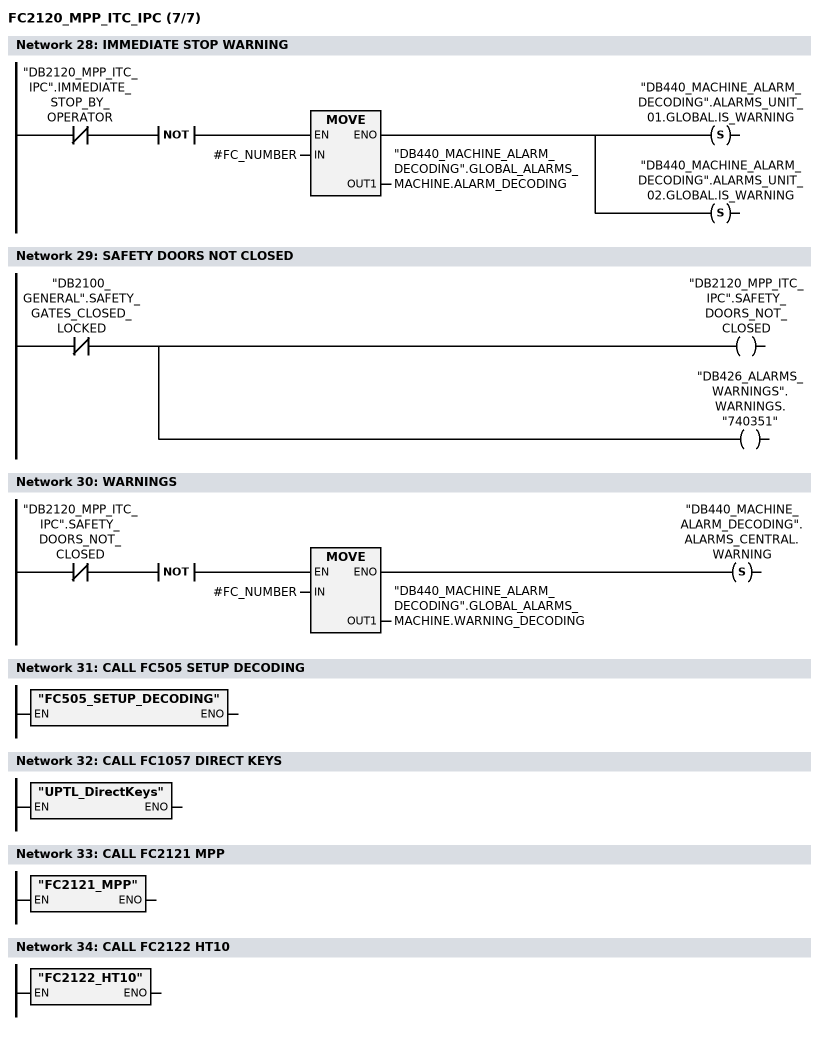
   RUNG wire#powerrail
      I_Contact( "DB2120_MPP_ITC_IPC".IMMEDIATE_STOP_BY_OPERATOR )
      Not()
      { S7_GenerateENO := "TRUE" } Move(in := #FC_NUMBER, out1 => "DB440_MACHINE_ALARM_DECODING".GLOBAL_ALARMS_MACHINE.ALARM_DECODING)
      wire#w1
      S_Coil( "DB440_MACHINE_ALARM_DECODING".ALARMS_UNIT_01.GLOBAL.IS_WARNING )
   END_RUNG
   RUNG wire#w1
      S_Coil( "DB440_MACHINE_ALARM_DECODING".ALARMS_UNIT_02.GLOBAL.IS_WARNING )
   END_RUNG
   // the same network as SCL:
   // ENO of a box is taken as its EN; it also drops when the box reports an error
   IF NOT (NOT "DB2120_MPP_ITC_IPC".IMMEDIATE_STOP_BY_OPERATOR) THEN
       "DB440_MACHINE_ALARM_DECODING".GLOBAL_ALARMS_MACHINE.ALARM_DECODING := #FC_NUMBER;
       "DB440_MACHINE_ALARM_DECODING".ALARMS_UNIT_01.GLOBAL.IS_WARNING := TRUE;
       "DB440_MACHINE_ALARM_DECODING".ALARMS_UNIT_02.GLOBAL.IS_WARNING := TRUE;
   END_IF;
END_REGION

REGION Network 29: SAFETY DOORS NOT CLOSED
   RUNG wire#powerrail
      I_Contact( "DB2100_GENERAL".SAFETY_GATES_CLOSED_LOCKED )
      wire#w1
      Coil( "DB2120_MPP_ITC_IPC".SAFETY_DOORS_NOT_CLOSED )
   END_RUNG
   RUNG wire#w1
      Coil( "DB426_ALARMS_WARNINGS".WARNINGS."740351" )
   END_RUNG
   // the same network as SCL:
   "DB2120_MPP_ITC_IPC".SAFETY_DOORS_NOT_CLOSED := NOT "DB2100_GENERAL".SAFETY_GATES_CLOSED_LOCKED;
   "DB426_ALARMS_WARNINGS".WARNINGS."740351" := NOT "DB2100_GENERAL".SAFETY_GATES_CLOSED_LOCKED;
END_REGION

REGION Network 30: WARNINGS
   RUNG wire#powerrail
      I_Contact( "DB2120_MPP_ITC_IPC".SAFETY_DOORS_NOT_CLOSED )
      Not()
      { S7_GenerateENO := "TRUE" } Move(in := #FC_NUMBER, out1 => "DB440_MACHINE_ALARM_DECODING".GLOBAL_ALARMS_MACHINE.WARNING_DECODING)
      S_Coil( "DB440_MACHINE_ALARM_DECODING".ALARMS_CENTRAL.WARNING )
   END_RUNG
   // the same network as SCL:
   // ENO of a box is taken as its EN; it also drops when the box reports an error
   IF NOT (NOT "DB2120_MPP_ITC_IPC".SAFETY_DOORS_NOT_CLOSED) THEN
       "DB440_MACHINE_ALARM_DECODING".GLOBAL_ALARMS_MACHINE.WARNING_DECODING := #FC_NUMBER;
       "DB440_MACHINE_ALARM_DECODING".ALARMS_CENTRAL.WARNING := TRUE;
   END_IF;
END_REGION

REGION Network 31: CALL FC505 SETUP DECODING
   RUNG wire#powerrail
      "FC505_SETUP_DECODING"()
   END_RUNG
   // the same network as SCL:
   "FC505_SETUP_DECODING"();
END_REGION

REGION Network 32: CALL FC1057 DIRECT KEYS
   RUNG wire#powerrail
      "UPTL_DirectKeys"()
   END_RUNG
   // the same network as SCL:
   "UPTL_DirectKeys"();
END_REGION

REGION Network 33: CALL FC2121 MPP
   RUNG wire#powerrail
      "FC2121_MPP"()
   END_RUNG
   // the same network as SCL:
   "FC2121_MPP"();
END_REGION

REGION Network 34: CALL FC2122 HT10
   RUNG wire#powerrail
      "FC2122_HT10"()
   END_RUNG
   // the same network as SCL:
   "FC2122_HT10"();
END_REGION
END_FUNCTION
